Fanuc KAREL source: wusecartacc.kl

PROGRAM wusecartacc
%NOLOCKGROUP
VAR
  p : POSITION
  q : POSITION
  i : INTEGER
  r : REAL
BEGIN
  WITH $USE_CARTACC = TRUE MOVE TO p
END wusecartacc
